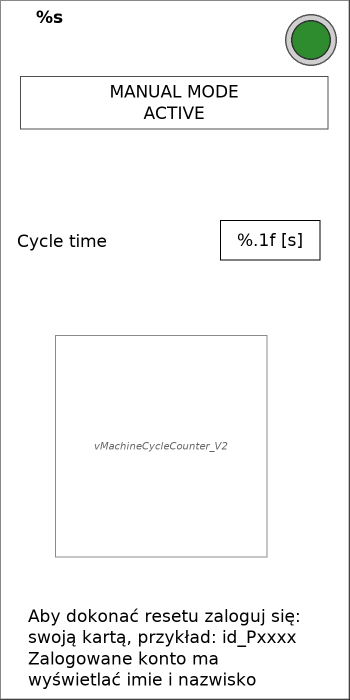
VISUALIZATION vHP3_Hp_Overview  // 350x700
VAR_IN_OUT
	fbHP	: fbHPv3_Control;
END_VAR
    RoundedRectangle (0,0 350x700)
    Lamp1 (281,10 60x60), variable: fbHP.stInOuts.bQ_LedTower_Blue, invisible if: NOT fbHP.stInOuts.bQ_LedTower_Blue, style: Lamp-Lamp1-Blue
    Lamp1 (281,10 60x60), variable: fbHP.stInOuts.bQ_LedTower_Yellow, invisible if: NOT fbHP.stInOuts.bQ_LedTower_Yellow, style: Lamp-Lamp1-Yellow
    Lamp1 (281,10 60x60), variable: fbHP.stInOuts.bQ_LedTower_Red, invisible if: NOT fbHP.stInOuts.bQ_LedTower_Red, style: Lamp-Lamp1-Red
    Lamp1 (281,10 60x60), variable: fbHP.stInOuts.bQ_LedTower_Green, invisible if: NOT fbHP.stInOuts.bQ_LedTower_Green, style: Lamp-Lamp1-Green
    Label (14,221 204x40), "Cycle time"
    Rectangle (220,220 100x40), "%.1f [s]", text variable: fbHP.rCycleTime_s
    Rectangle (20,76 308x53), "MANUAL MODE ACTIVE", invisible if: NOT fbHP.bManualMode
    RoundedRectangle (33,2 240x30), "%s", text list: 'tlHPv3', text index: fbHP.iMachineNumber
    Label (25,605 316x86), "Aby dokonać resetu zaloguj się: swoją kartą, przykład: id_Pxxxx Zalogowane konto ma wyświetlać imie i nazwisko"
    Frame (55,335 212x222)
        shows vMachineCycleCounter_V2(fb := fbHP.fbCoverCounter)
END_VISUALIZATION

(* stored: Version 1.1.0.1, ProductVersion 3.1.4024.13
   Visu vHP3_Hp_Overview: Id {fccc0e57-7314-4123-af96-e5177c6d6f3d} *)
